// TwinCAT 3 PLC project PLC1
// ProgramVersion: 3.1.4023.0
// libraries:
//   Tc2_Standard, * (Beckhoff Automation GmbH)
//   Tc2_System, * (Beckhoff Automation GmbH)
//   Tc3_Module, * (Beckhoff Automation GmbH)
// project tree:
//   GVLs/ GVL_IO.TcGVL
//   / PlcTask.TcTTO
//   POUs/ MAIN.TcPOU, POU_1.TcPOU
// real-time tasks:
//   TASK PlcTask: cycle T#10ms, priority 20, ADS port 350
// I/O:
//   DEVICE Device 1 (EtherCAT), AmsNetId 192.168.0.10.2.1
//     Term 1 (EK1100-0008) [EK1100-0008 EtherCAT Coupler M8 (2A E-Bus)]
//       Term 2 (EL9410) [EL9410 E-Bus Power Supplier  (Diagnostics)]
//       Term 4 (EL6614) [EL6614 4 Port Switch (Ethernet, CoE)]
//   DEVICE ek9 (Iot Mqtt Controller)
//     Box 3 (Subscriber)
//   DEVICE Device 3 (Virtual-Ethernet)
//     Box 5 (BC9020)
//     Box 6 (BK9000)

CONFIGURATION PLC1
    RESOURCE PLC ON TwinCAT3
        TASK PlcTask(INTERVAL := T#10ms, PRIORITY := 20);
        PROGRAM MAIN WITH PlcTask : MAIN;
        PROGRAM POU_1 WITH PlcTask : POU_1;
    END_RESOURCE
END_CONFIGURATION

// ---- GVLs/GVL_IO.TcGVL
//{attribute 'qualified_only'}
VAR_GLOBAL
	bPrzycisk1		AT%I*	:	BOOL;
	bPrzycisk2 		AT%I*	:	BOOL;
	bPrzycisk3		AT%I*	:	BOOL;
	bPrzycisk4		AT%I*	:	BOOL;
	
	bLampka1		AT%Q*	:	BOOL;
	bLampka2		AT%Q*	:	BOOL;
	bLampka3		AT%Q*	:	BOOL;
	bLampka4		AT%Q*	:	BOOL;

	iPotencjometr1	AT%I*	:	INT;
	iPotencjometr2	AT%I*	:	INT;
	
	iWyswietlacz1	AT%Q*	:	INT;
	iWyswietlacz2	AT%Q*	:	INT;
	
	
END_VAR

// ---- POUs/MAIN.TcPOU
PROGRAM MAIN
VAR
END_VAR

END_PROGRAM

// ---- POUs/POU_1.TcPOU
PROGRAM POU_1
VAR
	tCzas: TIME := T#3S;
	TON1: TON;
	TON2: TON;
END_VAR

TON1(IN := GVL_IO.bPrzycisk2, PT := tCzas); // TON
GVL_IO.bLampka3 := TON1.Q;
TON2(IN := TON1.Q, PT := 2*tCzas); // TON
GVL_IO.bLampka4 := TON2.Q;

END_PROGRAM
